TYPE TcoInsightUserData_v_5_x_x : STRUCT
    UserData AT %Q* : ARRAY[0..253] OF BYTE;
END_STRUCT
END_TYPE

(* stored: Version 1.1.0.1, ProductVersion 3.1.4024.11
   DUT TcoInsightUserData_v_5_x_x: Id {4424139a-d997-0a54-04e1-f7d23d8e6994} *)
